FUNCTION_BLOCK BACnetServer (* Service Interface Function Block Type *)
  (* Standard: 61499-2 *)
  (* Version 1.0, 2020-02-02, root *)
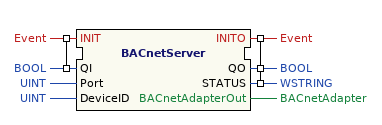
  EVENT_INPUT
    INIT WITH QI; (* Service Initialization *)
  END_EVENT
  EVENT_OUTPUT
    INITO WITH QO, STATUS; (* Initialization Confirm *)
  END_EVENT
  VAR_INPUT
    QI : BOOL; (* Event Input Qualifier *)
    Port : UINT; (* UDP Port number of the communication socket *)
    DeviceID : UINT; (* Identifier of the server's Device Object *)
  END_VAR
  VAR_OUTPUT
    QO : BOOL; (* Event Output Qualifier *)
    STATUS : WSTRING; (* Service Status *)
  END_VAR
  PLUGS
    BACnetAdapterOut : BACnetAdapter; (* BACnet adapter plug *)
  END_PLUGS
END_FUNCTION_BLOCK
